// TIA Portal V16 export
// export: Created 2021-11-12T13:32:30.3690276Z, ExportSetting WithDefaults, DisplayName Totally Integrated Automation Portal, DisplayVersion V16 Update 3, DisplayName TIA Portal Version Control Interface, DisplayVersion V16 Update 2, DisplayName TIA Portal Openness, DisplayVersion V16 Update 3, DisplayName SINAMICS Startdrive Advanced, DisplayVersion V16 Update 5, DisplayName SINAMICS Startdrive G130, G150, S120, S150, SINAMICS MV, S210, DisplayVersion V16 Update 5, DisplayName SINAMICS Startdrive G110M, G120, G120C, G120D, G120P, G115D, DisplayVersion V16 Update 5, DisplayName STEP 7 Professional, DisplayVersion V16 Update 3, DisplayName STEP 7 Safety, DisplayVersion V16, DisplayName WinCC UA Professional, DisplayVersion V16 Update 3
FUNCTION_BLOCK "Station 1R4 Seq"   // FB70, LAD
TITLE = Sequence
{ S7_Optimized_Access := 'TRUE' }
VERSION : 0.1
// MICE standard block 
// Sequence
// Block is designed as a template fo creating user sequences
// 
// All temp variables ToChangeXXXX should be replaced or removed.
// 
// Version              Created                        by             Comment
// 0.1                      30. 8. 2018                    PJ           initial version
// stored: AutoNumber true, IsIECCheckEnabled false, IsRetainMemResEnabled false, MemoryReserve 100, SetENOAutomatically false, UDAEnableTagReadback false
   VAR_INPUT
      IS_ZoneM { ExternalAccessible := 'False'; ExternalVisible := 'False'; ExternalWritable := 'False'} : "UDT_Status_main";   // Main structure from zone
      IS_ZoneS { ExternalAccessible := 'False'; ExternalVisible := 'False'; ExternalWritable := 'False'} : "UDT_Zone_Status_specific";   // Specific structure from zone
      IB1EnableSeq : Bool;   // Enable transition of sequence steps.
      IB1Init : Bool;   // Request to initialize sequence
      IB1SetStep : Bool;   // Request to set specific step number
      II_ReqStepNr : UInt;   // Specific step number to be set
      IB1AlmSupp : Bool;   // Alarm suppression - external
      IB1ExtError : Bool;   // External error
   END_VAR
   VAR_OUTPUT
      OS_Status : Struct   // Output status
         Main : "UDT_Status_main";
         Specific : "UDT_Sequence_Status_Specific";
         Error : "UDT_Error01";
      END_STRUCT;
   END_VAR
   VAR_IN_OUT
      XS_Parameter : "UDT_Sequence_Parameter";   // Individual parameter structure
      XS_Command : "UDT_Sequence_Command";   // Individual command structure
   END_VAR
   VAR RETAIN
      SS_Alarm : Struct   // Device alarms
         ExtError : Bool;   // External error / Externí porucha
         StepOvertime : Bool;   // Current step active for too long / Povolená doba trvání kroku překročena
         Res_0_2 : Bool;   // Reserve
         Res_0_3 : Bool;   // Reserve
         Res_0_4 : Bool;   // Reserve
         Res_0_5 : Bool;   // Reserve
         Res_0_6 : Bool;   // Reserve
         Res_0_7 : Bool;   // Reserve
      END_STRUCT;
   END_VAR
   VAR
      SS_Warning : Struct   // Device warnings
         Res : Bool;   // Reserve / Čeká se až bude signál v 1
         Res_1 : Bool;   // Reserve / Čeká se až bude signál v 0
         Res_2 : Bool;   // Reserve / Čeká se až bude signál v 1
         Res_3 : Bool;   // Reserve / Čeká se až bude signál v 0
         Res_4 : Bool;   // Reserve
         Res_5 : Bool;   // Reserve
         Res_6 : Bool;   // Reserve
         Res_7 : Bool;   // Reserve
      END_STRUCT;
      SB1CollErr : Bool;   // Collective error
      SB1CollWrn : Bool;   // Collective warning
   END_VAR
   VAR RETAIN
      SI_ActiveStepNr : UInt;   // Number of active step
   END_VAR
   VAR
      SI_PreviousStepNr : UInt;   // Number of previous step
      ST_TONStepDuration { S7_SetPoint := 'True'} : IEC_TIMER;   // Checking if step is not active for too long.
   END_VAR
   VAR_TEMP
      TS_Parameter : "UDT_Sequence_Parameter";
      TS_Command : "UDT_Sequence_Command";
      TS_Status : Struct
         Main : "UDT_Status_main";
         Specific : "UDT_Sequence_Status_Specific";
         Error : "UDT_Error01";
      END_STRUCT;
      TB1TransitionEnable : Bool;   // Condition from mode enable transition between steps
      TB1AlmSupp : Bool;   // Alarm suppression
      TI_StepTimeIndex : UInt;   // Index to find time for active step.
   END_VAR
   VAR_TEMP   // added for the SCL form of the ladder/FBD networks
      _w1 : Bool;
   END_VAR
BEGIN

REGION Network 1: Clear temporary variables TS_Status - Main, Specific
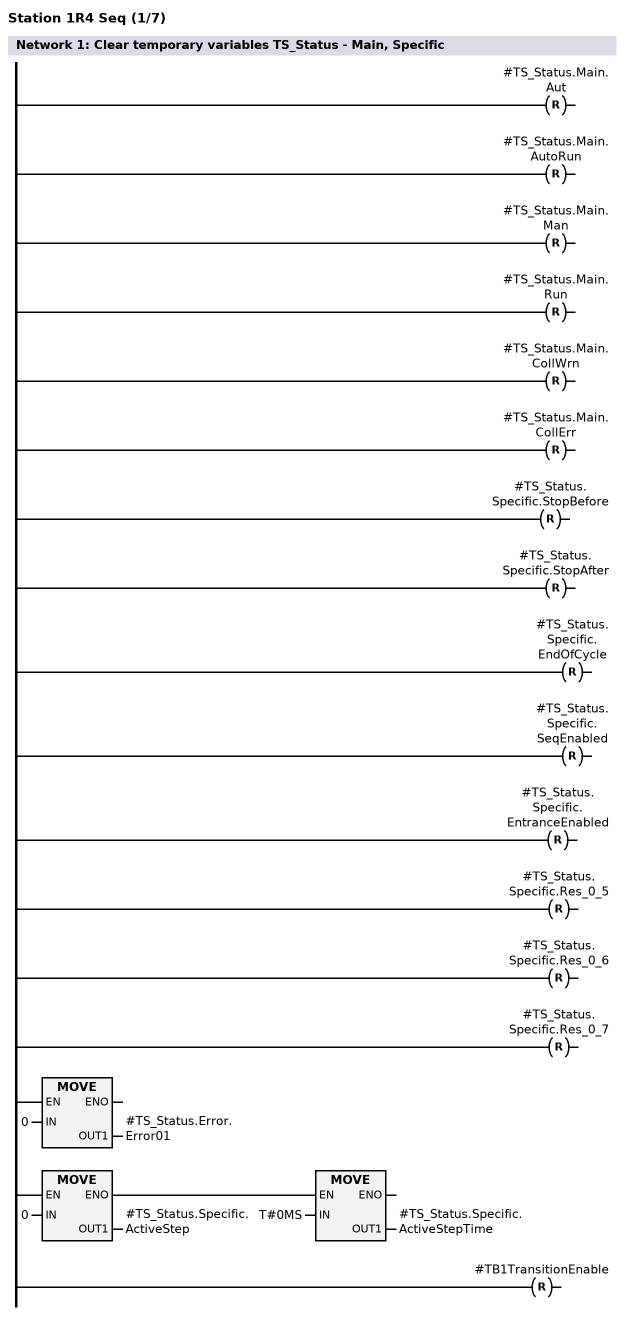
   RUNG wire#powerrail
      R_Coil( #TS_Status.Main.Aut )
   END_RUNG
   RUNG wire#powerrail
      R_Coil( #TS_Status.Main.AutoRun )
   END_RUNG
   RUNG wire#powerrail
      R_Coil( #TS_Status.Main.Man )
   END_RUNG
   RUNG wire#powerrail
      R_Coil( #TS_Status.Main.Run )
   END_RUNG
   RUNG wire#powerrail
      R_Coil( #TS_Status.Main.CollWrn )
   END_RUNG
   RUNG wire#powerrail
      R_Coil( #TS_Status.Main.CollErr )
   END_RUNG
   RUNG wire#powerrail
      R_Coil( #TS_Status.Specific.StopBefore )
   END_RUNG
   RUNG wire#powerrail
      R_Coil( #TS_Status.Specific.StopAfter )
   END_RUNG
   RUNG wire#powerrail
      R_Coil( #TS_Status.Specific.EndOfCycle )
   END_RUNG
   RUNG wire#powerrail
      R_Coil( #TS_Status.Specific.SeqEnabled )
   END_RUNG
   RUNG wire#powerrail
      R_Coil( #TS_Status.Specific.EntranceEnabled )
   END_RUNG
   RUNG wire#powerrail
      R_Coil( #TS_Status.Specific.Res_0_5 )
   END_RUNG
   RUNG wire#powerrail
      R_Coil( #TS_Status.Specific.Res_0_6 )
   END_RUNG
   RUNG wire#powerrail
      R_Coil( #TS_Status.Specific.Res_0_7 )
   END_RUNG
   RUNG wire#powerrail
      Move(in := 0, out1 => #TS_Status.Error.Error01)
   END_RUNG
   RUNG wire#powerrail
      Move(in := 0, out1 => #TS_Status.Specific.ActiveStep)
      Move(in := T#0MS, out1 => #TS_Status.Specific.ActiveStepTime)
   END_RUNG
   RUNG wire#powerrail
      R_Coil( #TB1TransitionEnable )
   END_RUNG
   // the same network as SCL:
   #TS_Status.Main.Aut := FALSE;
   #TS_Status.Main.AutoRun := FALSE;
   #TS_Status.Main.Man := FALSE;
   #TS_Status.Main.Run := FALSE;
   #TS_Status.Main.CollWrn := FALSE;
   #TS_Status.Main.CollErr := FALSE;
   #TS_Status.Specific.StopBefore := FALSE;
   #TS_Status.Specific.StopAfter := FALSE;
   #TS_Status.Specific.EndOfCycle := FALSE;
   #TS_Status.Specific.SeqEnabled := FALSE;
   #TS_Status.Specific.EntranceEnabled := FALSE;
   #TS_Status.Specific.Res_0_5 := FALSE;
   #TS_Status.Specific.Res_0_6 := FALSE;
   #TS_Status.Specific.Res_0_7 := FALSE;
   #TS_Status.Error.Error01 := 0;
   #TS_Status.Specific.ActiveStep := 0;
   #TS_Status.Specific.ActiveStepTime := T#0MS;
   #TB1TransitionEnable := FALSE;
END_REGION

REGION Network 2: Copy In/Out variables to temporary variables
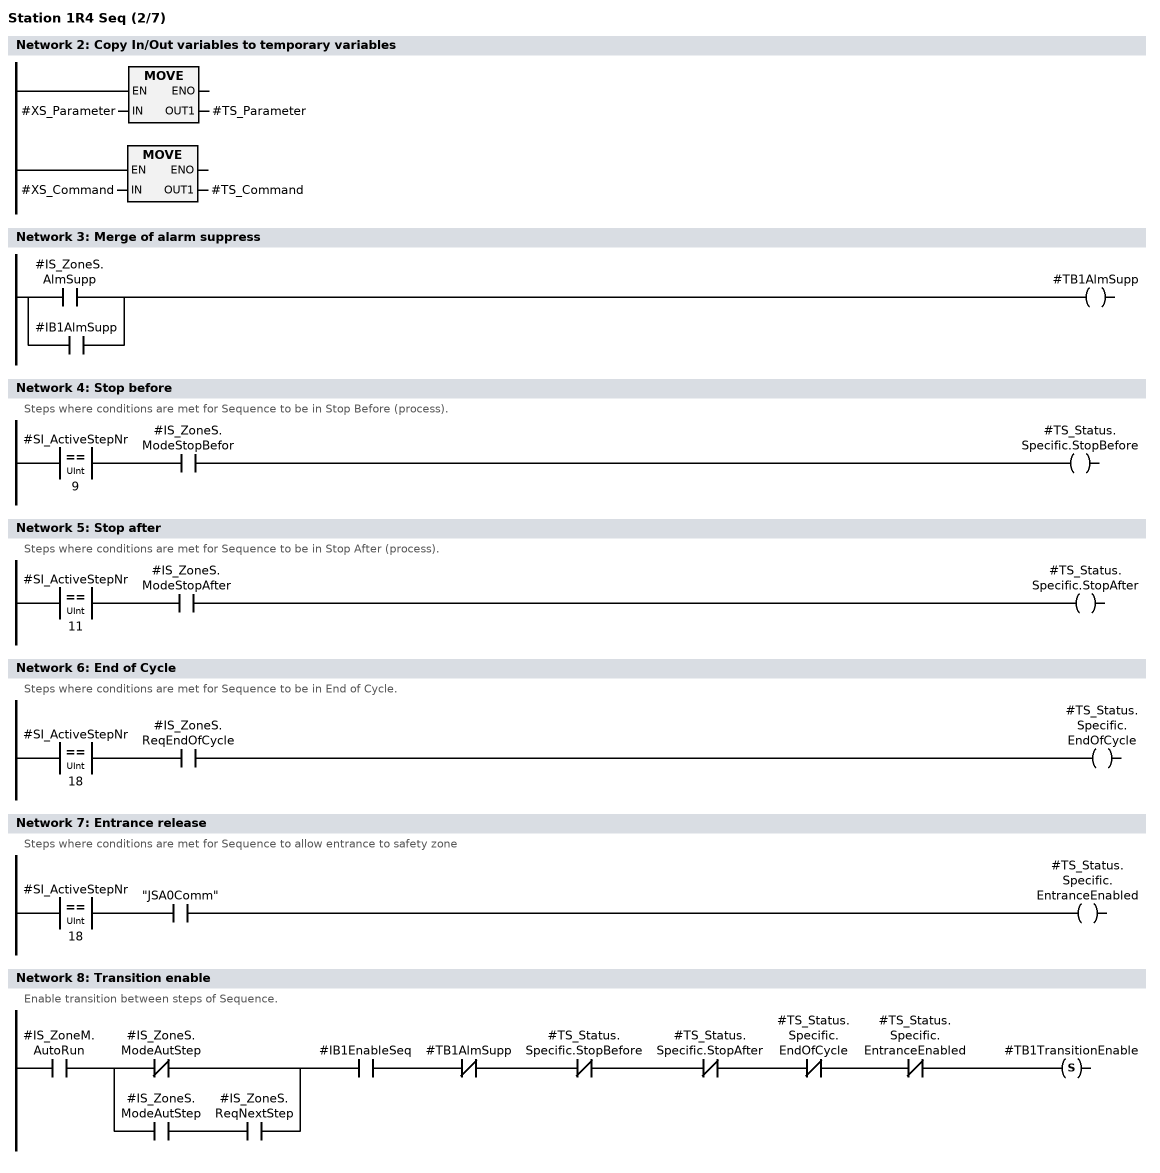
   RUNG wire#powerrail
      Move(in := #XS_Parameter, out1 => #TS_Parameter)
   END_RUNG
   RUNG wire#powerrail
      Move(in := #XS_Command, out1 => #TS_Command)
   END_RUNG
   // the same network as SCL:
   #TS_Parameter := #XS_Parameter;
   #TS_Command := #XS_Command;
END_REGION

REGION Network 3: Merge of alarm suppress
   RUNG wire#powerrail
      Contact( #IS_ZoneS.AlmSupp )
      wire#w1
      Coil( #TB1AlmSupp )
   END_RUNG
   RUNG wire#powerrail
      Contact( #IB1AlmSupp )
   END_RUNG wire#w1
   // the same network as SCL:
   #TB1AlmSupp := #IS_ZoneS.AlmSupp OR #IB1AlmSupp;
END_REGION

REGION Network 4: Stop before
   // Steps where conditions are met for Sequence to be in Stop Before (process).
   RUNG wire#powerrail
      { S7_Templates := "SrcType := UInt" } EQ_Contact(in1 := #SI_ActiveStepNr, in2 := 9)
      Contact( #IS_ZoneS.ModeStopBefor )
      Coil( #TS_Status.Specific.StopBefore )
   END_RUNG
   // the same network as SCL:
   #TS_Status.Specific.StopBefore := (#SI_ActiveStepNr = 9) AND #IS_ZoneS.ModeStopBefor;
END_REGION

REGION Network 5: Stop after
   // Steps where conditions are met for Sequence to be in Stop After (process).
   RUNG wire#powerrail
      { S7_Templates := "SrcType := UInt" } EQ_Contact(in1 := #SI_ActiveStepNr, in2 := 11)
      Contact( #IS_ZoneS.ModeStopAfter )
      Coil( #TS_Status.Specific.StopAfter )
   END_RUNG
   // the same network as SCL:
   #TS_Status.Specific.StopAfter := (#SI_ActiveStepNr = 11) AND #IS_ZoneS.ModeStopAfter;
END_REGION

REGION Network 6: End of Cycle
   // Steps where conditions are met for Sequence to be in End of Cycle.
   RUNG wire#powerrail
      { S7_Templates := "SrcType := UInt" } EQ_Contact(in1 := #SI_ActiveStepNr, in2 := 18)
      Contact( #IS_ZoneS.ReqEndOfCycle )
      Coil( #TS_Status.Specific.EndOfCycle )
   END_RUNG
   // the same network as SCL:
   #TS_Status.Specific.EndOfCycle := (#SI_ActiveStepNr = 18) AND #IS_ZoneS.ReqEndOfCycle;
END_REGION

REGION Network 7: Entrance release
   // Steps where conditions are met for Sequence to allow entrance to safety zone
   RUNG wire#powerrail
      { S7_Templates := "SrcType := UInt" } EQ_Contact(in1 := #SI_ActiveStepNr, in2 := 18)
      Contact( "JSA0Comm" )
      Coil( #TS_Status.Specific.EntranceEnabled )
   END_RUNG
   // the same network as SCL:
   #TS_Status.Specific.EntranceEnabled := (#SI_ActiveStepNr = 18) AND "JSA0Comm";
END_REGION

REGION Network 8: Transition enable
   // Enable transition between steps of Sequence.
   RUNG wire#powerrail
      Contact( #IS_ZoneM.AutoRun )
      wire#w1
      I_Contact( #IS_ZoneS.ModeAutStep )
      wire#w2
      Contact( #IB1EnableSeq )
      I_Contact( #TB1AlmSupp )
      I_Contact( #TS_Status.Specific.StopBefore )
      I_Contact( #TS_Status.Specific.StopAfter )
      I_Contact( #TS_Status.Specific.EndOfCycle )
      I_Contact( #TS_Status.Specific.EntranceEnabled )
      S_Coil( #TB1TransitionEnable )
   END_RUNG
   RUNG wire#w1
      Contact( #IS_ZoneS.ModeAutStep )
      Contact( #IS_ZoneS.ReqNextStep )
   END_RUNG wire#w2
   // the same network as SCL:
   IF #IS_ZoneM.AutoRun AND (NOT #IS_ZoneS.ModeAutStep OR (#IS_ZoneS.ModeAutStep AND #IS_ZoneS.ReqNextStep)) AND #IB1EnableSeq AND NOT #TB1AlmSupp AND NOT #TS_Status.Specific.StopBefore AND NOT #TS_Status.Specific.StopAfter AND NOT #TS_Status.Specific.EndOfCycle AND NOT #TS_Status.Specific.EntranceEnabled THEN
       #TB1TransitionEnable := TRUE;
   END_IF;
END_REGION

REGION Network 9: Init sequence
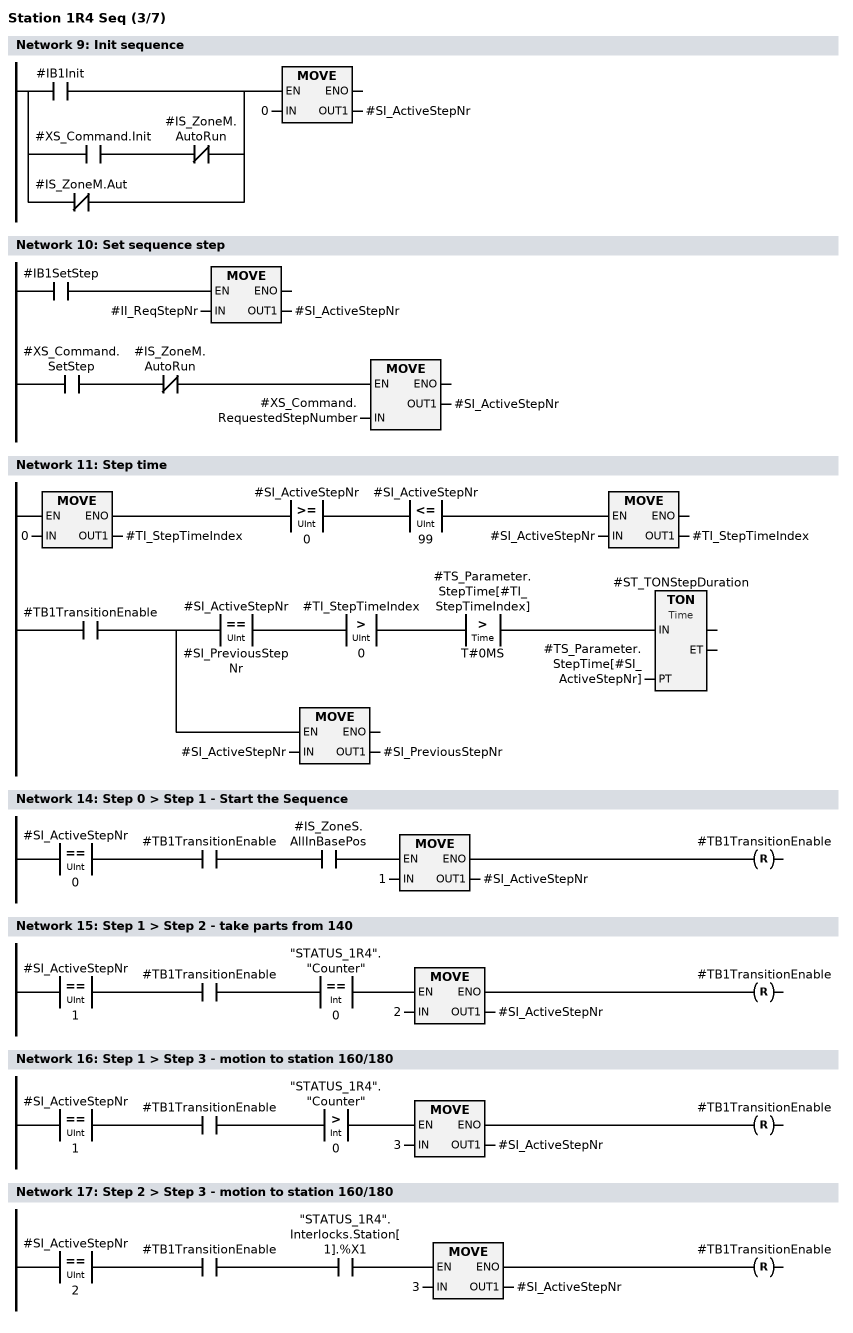
   RUNG wire#powerrail
      Contact( #IB1Init )
      wire#w1
      Move(in := 0, out1 => #SI_ActiveStepNr)
   END_RUNG
   RUNG wire#powerrail
      Contact( #XS_Command.Init )
      I_Contact( #IS_ZoneM.AutoRun )
   END_RUNG wire#w1
   RUNG wire#powerrail
      I_Contact( #IS_ZoneM.Aut )
   END_RUNG wire#w1
   // the same network as SCL:
   IF #IB1Init OR (#XS_Command.Init AND NOT #IS_ZoneM.AutoRun) OR NOT #IS_ZoneM.Aut THEN
       #SI_ActiveStepNr := 0;
   END_IF;
END_REGION

REGION Network 10: Set sequence step
   RUNG wire#powerrail
      Contact( #IB1SetStep )
      Move(in := #II_ReqStepNr, out1 => #SI_ActiveStepNr)
   END_RUNG
   RUNG wire#powerrail
      Contact( #XS_Command.SetStep )
      I_Contact( #IS_ZoneM.AutoRun )
      Move(in := #XS_Command.RequestedStepNumber, out1 => #SI_ActiveStepNr)
   END_RUNG
   // the same network as SCL:
   IF #IB1SetStep THEN #SI_ActiveStepNr := #II_ReqStepNr; END_IF;
   IF #XS_Command.SetStep AND NOT #IS_ZoneM.AutoRun THEN
       #SI_ActiveStepNr := #XS_Command.RequestedStepNumber;
   END_IF;
END_REGION

REGION Network 11: Step time
   RUNG wire#powerrail
      Move(in := 0, out1 => #TI_StepTimeIndex)
      { S7_Templates := "SrcType := UInt" } GE_Contact(in1 := #SI_ActiveStepNr, in2 := 0)
      { S7_Templates := "SrcType := UInt" } LE_Contact(in1 := #SI_ActiveStepNr, in2 := 99)
      Move(in := #SI_ActiveStepNr, out1 => #TI_StepTimeIndex)
   END_RUNG
   RUNG wire#powerrail
      Contact( #TB1TransitionEnable )
      wire#w1
      { S7_Templates := "SrcType := UInt" } EQ_Contact(in1 := #SI_ActiveStepNr, in2 := #SI_PreviousStepNr)
      { S7_Templates := "SrcType := UInt" } GT_Contact(in1 := #TI_StepTimeIndex, in2 := 0)
      { S7_Templates := "SrcType := Time" } GT_Contact(in1 := #TS_Parameter.StepTime[#TI_StepTimeIndex], in2 := T#0MS)
      { S7_Templates := "time_type := Time" } #ST_TONStepDuration.TON(pt := #TS_Parameter.StepTime[#SI_ActiveStepNr], et =>)
   END_RUNG
   RUNG wire#w1
      Move(in := #SI_ActiveStepNr, out1 => #SI_PreviousStepNr)
   END_RUNG
   // the same network as SCL:
   #TI_StepTimeIndex := 0;
   IF (#SI_ActiveStepNr >= 0) AND (#SI_ActiveStepNr <= 99) THEN
       #TI_StepTimeIndex := #SI_ActiveStepNr;
   END_IF;
   #ST_TONStepDuration.TON(IN := #TB1TransitionEnable AND (#SI_ActiveStepNr = #SI_PreviousStepNr) AND (#TI_StepTimeIndex > 0) AND (#TS_Parameter.StepTime[#TI_StepTimeIndex] > T#0MS),
                           PT := #TS_Parameter.StepTime[#SI_ActiveStepNr]);
   IF #TB1TransitionEnable THEN #SI_PreviousStepNr := #SI_ActiveStepNr; END_IF;
END_REGION

REGION Network 12: Operator info status
END_REGION

REGION Network 13: *************** Sequence steps ***********************
   // No parallel conditions. If neccessary > for each condition its own network (Active step / conditions / step change). This also solves jumps.
   // No "active" parts in step. So no timers, counters, comparators etc. those belong to Creating conditions section or outside this block. Only simple bool conditions.
   // Always reset TB1_TransitionEnable bit. This will make sure on PLC cycle only one step of sequence will be processed.
   // Last step/network should be that if active step number is bigger then last used one go to zero step.
END_REGION

REGION Network 14: Step 0 > Step 1 - Start the Sequence
   RUNG wire#powerrail
      { S7_Templates := "SrcType := UInt" } EQ_Contact(in1 := #SI_ActiveStepNr, in2 := 0)
      Contact( #TB1TransitionEnable )
      Contact( #IS_ZoneS.AllInBasePos )
      Move(in := 1, out1 => #SI_ActiveStepNr)
      R_Coil( #TB1TransitionEnable )
   END_RUNG
   // the same network as SCL:
   #_w1 := (#SI_ActiveStepNr = 0) AND #TB1TransitionEnable AND #IS_ZoneS.AllInBasePos;
   IF #_w1 THEN
       #SI_ActiveStepNr := 1;
       #TB1TransitionEnable := FALSE;
   END_IF;
END_REGION

REGION Network 15: Step 1 > Step 2 - take parts from 140
   RUNG wire#powerrail
      { S7_Templates := "SrcType := UInt" } EQ_Contact(in1 := #SI_ActiveStepNr, in2 := 1)
      Contact( #TB1TransitionEnable )
      { S7_Templates := "SrcType := Int" } EQ_Contact(in1 := "STATUS_1R4"."Counter", in2 := 0)
      Move(in := 2, out1 => #SI_ActiveStepNr)
      R_Coil( #TB1TransitionEnable )
   END_RUNG
   // the same network as SCL:
   #_w1 := (#SI_ActiveStepNr = 1) AND #TB1TransitionEnable AND ("STATUS_1R4"."Counter" = 0);
   IF #_w1 THEN
       #SI_ActiveStepNr := 2;
       #TB1TransitionEnable := FALSE;
   END_IF;
END_REGION

REGION Network 16: Step 1 > Step 3 - motion to station 160/180
   RUNG wire#powerrail
      { S7_Templates := "SrcType := UInt" } EQ_Contact(in1 := #SI_ActiveStepNr, in2 := 1)
      Contact( #TB1TransitionEnable )
      { S7_Templates := "SrcType := Int" } GT_Contact(in1 := "STATUS_1R4"."Counter", in2 := 0)
      Move(in := 3, out1 => #SI_ActiveStepNr)
      R_Coil( #TB1TransitionEnable )
   END_RUNG
   // the same network as SCL:
   #_w1 := (#SI_ActiveStepNr = 1) AND #TB1TransitionEnable AND ("STATUS_1R4"."Counter" > 0);
   IF #_w1 THEN
       #SI_ActiveStepNr := 3;
       #TB1TransitionEnable := FALSE;
   END_IF;
END_REGION

REGION Network 17: Step 2 > Step 3 - motion to station 160/180
   RUNG wire#powerrail
      { S7_Templates := "SrcType := UInt" } EQ_Contact(in1 := #SI_ActiveStepNr, in2 := 2)
      Contact( #TB1TransitionEnable )
      Contact( "STATUS_1R4".Interlocks.Station[1].%X1 )
      Move(in := 3, out1 => #SI_ActiveStepNr)
      R_Coil( #TB1TransitionEnable )
   END_RUNG
   // the same network as SCL:
   #_w1 := (#SI_ActiveStepNr = 2) AND #TB1TransitionEnable AND "STATUS_1R4".Interlocks.Station[1].%X1;
   IF #_w1 THEN
       #SI_ActiveStepNr := 3;
       #TB1TransitionEnable := FALSE;
   END_IF;
END_REGION

REGION Network 18: Step 3 > Step 4 - put parts to station 160 / 180
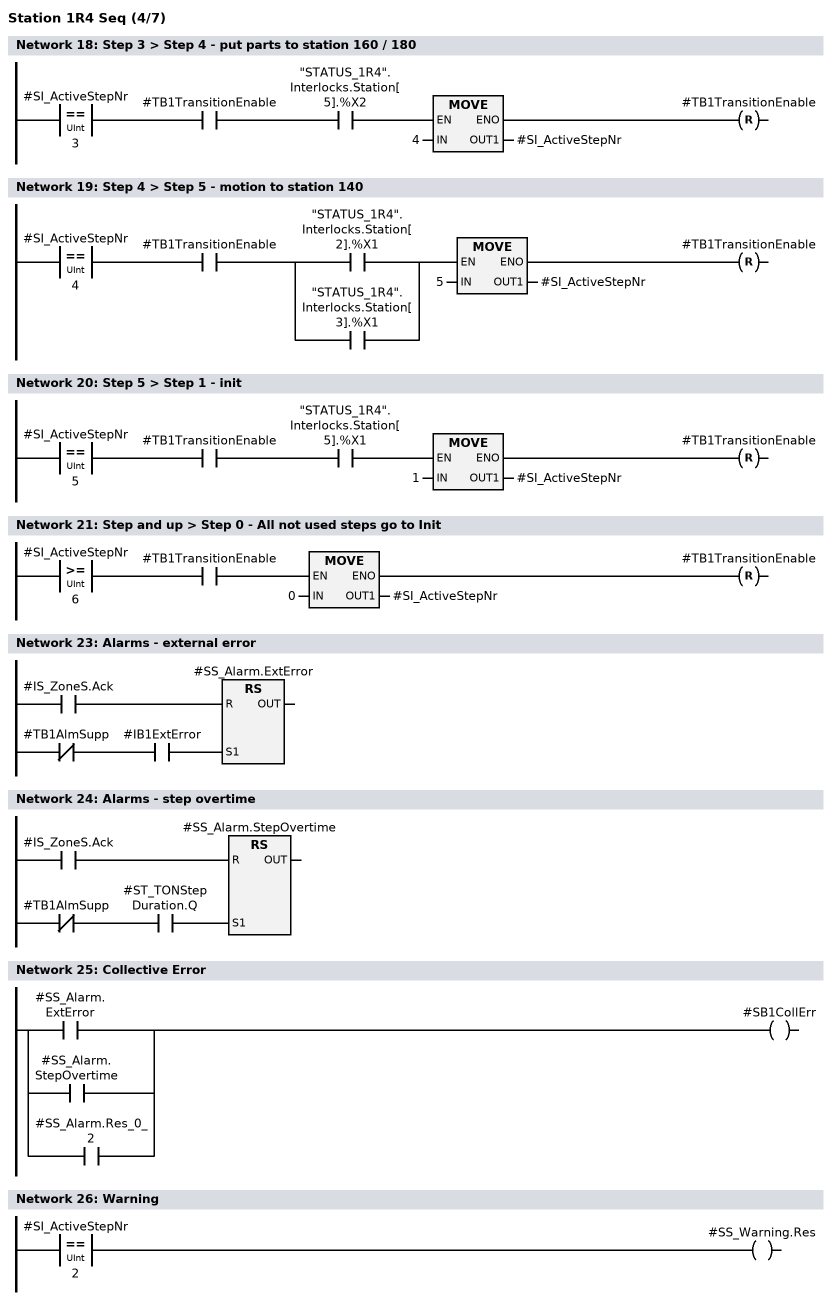
   RUNG wire#powerrail
      { S7_Templates := "SrcType := UInt" } EQ_Contact(in1 := #SI_ActiveStepNr, in2 := 3)
      Contact( #TB1TransitionEnable )
      Contact( "STATUS_1R4".Interlocks.Station[5].%X2 )
      Move(in := 4, out1 => #SI_ActiveStepNr)
      R_Coil( #TB1TransitionEnable )
   END_RUNG
   // the same network as SCL:
   #_w1 := (#SI_ActiveStepNr = 3) AND #TB1TransitionEnable AND "STATUS_1R4".Interlocks.Station[5].%X2;
   IF #_w1 THEN
       #SI_ActiveStepNr := 4;
       #TB1TransitionEnable := FALSE;
   END_IF;
END_REGION

REGION Network 19: Step 4 > Step 5 - motion to station 140
   RUNG wire#powerrail
      { S7_Templates := "SrcType := UInt" } EQ_Contact(in1 := #SI_ActiveStepNr, in2 := 4)
      Contact( #TB1TransitionEnable )
      wire#w1
      Contact( "STATUS_1R4".Interlocks.Station[2].%X1 )
      wire#w2
      Move(in := 5, out1 => #SI_ActiveStepNr)
      R_Coil( #TB1TransitionEnable )
   END_RUNG
   RUNG wire#w1
      Contact( "STATUS_1R4".Interlocks.Station[3].%X1 )
   END_RUNG wire#w2
   // the same network as SCL:
   #_w1 := (#SI_ActiveStepNr = 4) AND #TB1TransitionEnable AND ("STATUS_1R4".Interlocks.Station[2].%X1 OR "STATUS_1R4".Interlocks.Station[3].%X1);
   IF #_w1 THEN
       #SI_ActiveStepNr := 5;
       #TB1TransitionEnable := FALSE;
   END_IF;
END_REGION

REGION Network 20: Step 5 > Step 1 - init
   RUNG wire#powerrail
      { S7_Templates := "SrcType := UInt" } EQ_Contact(in1 := #SI_ActiveStepNr, in2 := 5)
      Contact( #TB1TransitionEnable )
      Contact( "STATUS_1R4".Interlocks.Station[5].%X1 )
      Move(in := 1, out1 => #SI_ActiveStepNr)
      R_Coil( #TB1TransitionEnable )
   END_RUNG
   // the same network as SCL:
   #_w1 := (#SI_ActiveStepNr = 5) AND #TB1TransitionEnable AND "STATUS_1R4".Interlocks.Station[5].%X1;
   IF #_w1 THEN
       #SI_ActiveStepNr := 1;
       #TB1TransitionEnable := FALSE;
   END_IF;
END_REGION

REGION Network 21: Step and up > Step 0 - All not used steps go to Init
   RUNG wire#powerrail
      { S7_Templates := "SrcType := UInt" } GE_Contact(in1 := #SI_ActiveStepNr, in2 := 6)
      Contact( #TB1TransitionEnable )
      Move(in := 0, out1 => #SI_ActiveStepNr)
      R_Coil( #TB1TransitionEnable )
   END_RUNG
   // the same network as SCL:
   #_w1 := (#SI_ActiveStepNr >= 6) AND #TB1TransitionEnable;
   IF #_w1 THEN
       #SI_ActiveStepNr := 0;
       #TB1TransitionEnable := FALSE;
   END_IF;
END_REGION

REGION Network 22: *************** Alarm and warning section ***********************
END_REGION

REGION Network 23: Alarms - external error
   RUNG wire#powerrail
      Contact( #IS_ZoneS.Ack )
      S_RS(operand := #SS_Alarm.ExtError, s1 := wire#w1)
   END_RUNG
   RUNG wire#powerrail
      I_Contact( #TB1AlmSupp )
      Contact( #IB1ExtError )
   END_RUNG wire#w1
   // the same network as SCL:
   IF #IS_ZoneS.Ack THEN
       #SS_Alarm.ExtError := FALSE;   // RS flip-flop
   END_IF;
   IF NOT #TB1AlmSupp AND #IB1ExtError THEN #SS_Alarm.ExtError := TRUE; END_IF;
END_REGION

REGION Network 24: Alarms - step overtime
   RUNG wire#powerrail
      Contact( #IS_ZoneS.Ack )
      S_RS(operand := #SS_Alarm.StepOvertime, s1 := wire#w1)
   END_RUNG
   RUNG wire#powerrail
      I_Contact( #TB1AlmSupp )
      Contact( #ST_TONStepDuration.Q )
   END_RUNG wire#w1
   // the same network as SCL:
   IF #IS_ZoneS.Ack THEN
       #SS_Alarm.StepOvertime := FALSE;   // RS flip-flop
   END_IF;
   IF NOT #TB1AlmSupp AND #ST_TONStepDuration.Q THEN #SS_Alarm.StepOvertime := TRUE; END_IF;
END_REGION

REGION Network 25: Collective Error
   RUNG wire#powerrail
      Contact( #SS_Alarm.ExtError )
      wire#w1
      Coil( #SB1CollErr )
   END_RUNG
   RUNG wire#powerrail
      Contact( #SS_Alarm.StepOvertime )
   END_RUNG wire#w1
   RUNG wire#powerrail
      Contact( #SS_Alarm.Res_0_2 )
   END_RUNG wire#w1
   // the same network as SCL:
   #SB1CollErr := #SS_Alarm.ExtError OR #SS_Alarm.StepOvertime OR #SS_Alarm.Res_0_2;
END_REGION

REGION Network 26: Warning
   RUNG wire#powerrail
      { S7_Templates := "SrcType := UInt" } EQ_Contact(in1 := #SI_ActiveStepNr, in2 := 2)
      Coil( #SS_Warning.Res )
   END_RUNG
   // the same network as SCL:
   #SS_Warning.Res := #SI_ActiveStepNr = 2;
END_REGION

REGION Network 27: Collective Warning
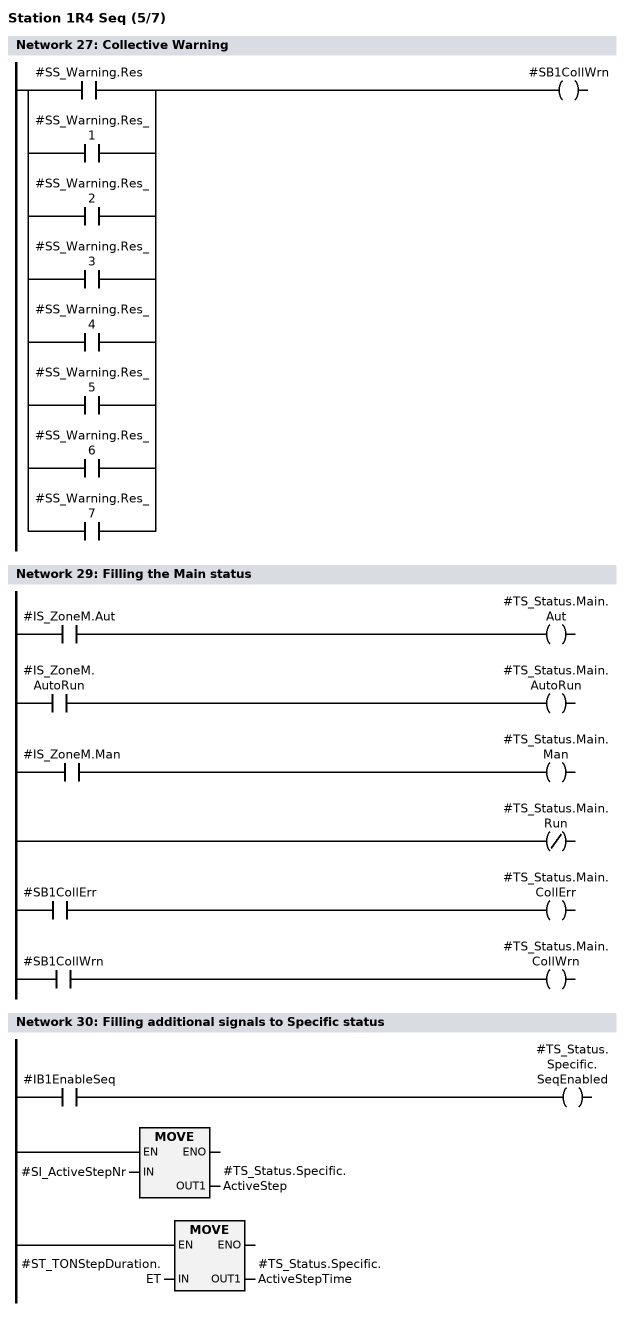
   RUNG wire#powerrail
      Contact( #SS_Warning.Res )
      wire#w1
      Coil( #SB1CollWrn )
   END_RUNG
   RUNG wire#powerrail
      Contact( #SS_Warning.Res_1 )
   END_RUNG wire#w1
   RUNG wire#powerrail
      Contact( #SS_Warning.Res_2 )
   END_RUNG wire#w1
   RUNG wire#powerrail
      Contact( #SS_Warning.Res_3 )
   END_RUNG wire#w1
   RUNG wire#powerrail
      Contact( #SS_Warning.Res_4 )
   END_RUNG wire#w1
   RUNG wire#powerrail
      Contact( #SS_Warning.Res_5 )
   END_RUNG wire#w1
   RUNG wire#powerrail
      Contact( #SS_Warning.Res_6 )
   END_RUNG wire#w1
   RUNG wire#powerrail
      Contact( #SS_Warning.Res_7 )
   END_RUNG wire#w1
   // the same network as SCL:
   #SB1CollWrn := #SS_Warning.Res OR #SS_Warning.Res_1 OR #SS_Warning.Res_2 OR #SS_Warning.Res_3 OR #SS_Warning.Res_4 OR #SS_Warning.Res_5 OR #SS_Warning.Res_6 OR #SS_Warning.Res_7;
END_REGION

REGION Network 28: *************** Fill out structures / Copy to outputs ***********************
END_REGION

REGION Network 29: Filling the Main status
   RUNG wire#powerrail
      Contact( #IS_ZoneM.Aut )
      Coil( #TS_Status.Main.Aut )
   END_RUNG
   RUNG wire#powerrail
      Contact( #IS_ZoneM.AutoRun )
      Coil( #TS_Status.Main.AutoRun )
   END_RUNG
   RUNG wire#powerrail
      Contact( #IS_ZoneM.Man )
      Coil( #TS_Status.Main.Man )
   END_RUNG
   RUNG wire#powerrail
      I_Coil( #TS_Status.Main.Run )
   END_RUNG
   RUNG wire#powerrail
      Contact( #SB1CollErr )
      Coil( #TS_Status.Main.CollErr )
   END_RUNG
   RUNG wire#powerrail
      Contact( #SB1CollWrn )
      Coil( #TS_Status.Main.CollWrn )
   END_RUNG
   // the same network as SCL:
   #TS_Status.Main.Aut := #IS_ZoneM.Aut;
   #TS_Status.Main.AutoRun := #IS_ZoneM.AutoRun;
   #TS_Status.Main.Man := #IS_ZoneM.Man;
   #TS_Status.Main.Run := NOT TRUE;
   #TS_Status.Main.CollErr := #SB1CollErr;
   #TS_Status.Main.CollWrn := #SB1CollWrn;
END_REGION

REGION Network 30: Filling additional signals to Specific status
   RUNG wire#powerrail
      Contact( #IB1EnableSeq )
      Coil( #TS_Status.Specific.SeqEnabled )
   END_RUNG
   RUNG wire#powerrail
      Move(in := #SI_ActiveStepNr, out1 => #TS_Status.Specific.ActiveStep)
   END_RUNG
   RUNG wire#powerrail
      Move(in := #ST_TONStepDuration.ET, out1 => #TS_Status.Specific.ActiveStepTime)
   END_RUNG
   // the same network as SCL:
   #TS_Status.Specific.SeqEnabled := #IB1EnableSeq;
   #TS_Status.Specific.ActiveStep := #SI_ActiveStepNr;
   #TS_Status.Specific.ActiveStepTime := #ST_TONStepDuration.ET;
END_REGION

REGION Network 31: Reset commands
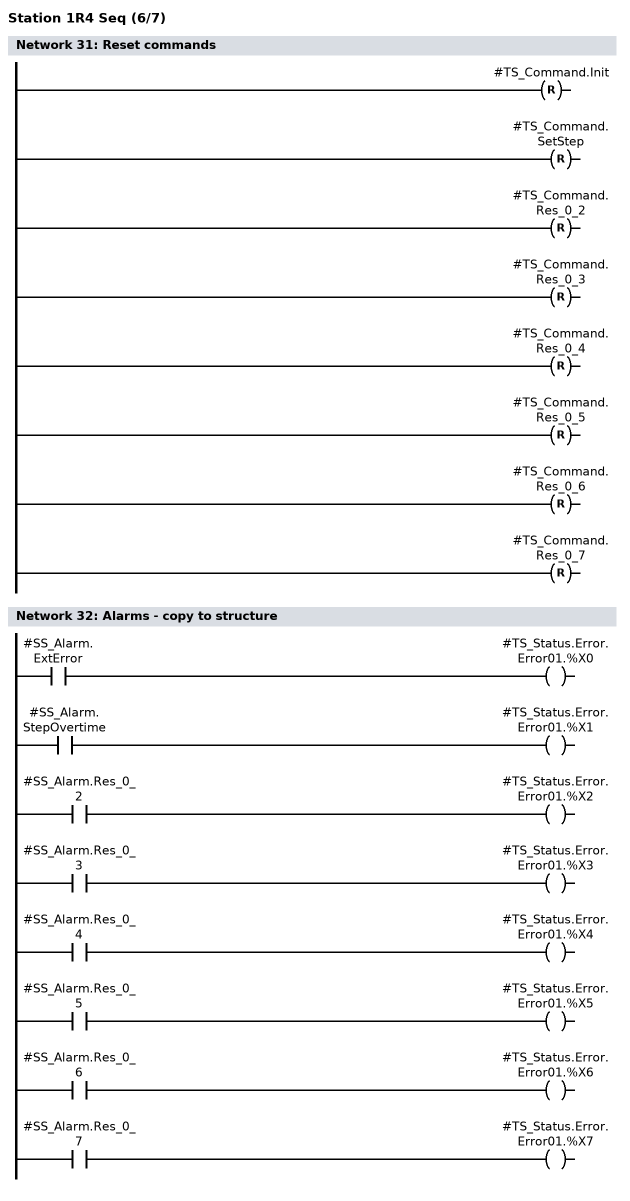
   RUNG wire#powerrail
      R_Coil( #TS_Command.Init )
   END_RUNG
   RUNG wire#powerrail
      R_Coil( #TS_Command.SetStep )
   END_RUNG
   RUNG wire#powerrail
      R_Coil( #TS_Command.Res_0_2 )
   END_RUNG
   RUNG wire#powerrail
      R_Coil( #TS_Command.Res_0_3 )
   END_RUNG
   RUNG wire#powerrail
      R_Coil( #TS_Command.Res_0_4 )
   END_RUNG
   RUNG wire#powerrail
      R_Coil( #TS_Command.Res_0_5 )
   END_RUNG
   RUNG wire#powerrail
      R_Coil( #TS_Command.Res_0_6 )
   END_RUNG
   RUNG wire#powerrail
      R_Coil( #TS_Command.Res_0_7 )
   END_RUNG
   // the same network as SCL:
   #TS_Command.Init := FALSE;
   #TS_Command.SetStep := FALSE;
   #TS_Command.Res_0_2 := FALSE;
   #TS_Command.Res_0_3 := FALSE;
   #TS_Command.Res_0_4 := FALSE;
   #TS_Command.Res_0_5 := FALSE;
   #TS_Command.Res_0_6 := FALSE;
   #TS_Command.Res_0_7 := FALSE;
END_REGION

REGION Network 32: Alarms - copy to structure
   RUNG wire#powerrail
      Contact( #SS_Alarm.ExtError )
      Coil( #TS_Status.Error.Error01.%X0 )
   END_RUNG
   RUNG wire#powerrail
      Contact( #SS_Alarm.StepOvertime )
      Coil( #TS_Status.Error.Error01.%X1 )
   END_RUNG
   RUNG wire#powerrail
      Contact( #SS_Alarm.Res_0_2 )
      Coil( #TS_Status.Error.Error01.%X2 )
   END_RUNG
   RUNG wire#powerrail
      Contact( #SS_Alarm.Res_0_3 )
      Coil( #TS_Status.Error.Error01.%X3 )
   END_RUNG
   RUNG wire#powerrail
      Contact( #SS_Alarm.Res_0_4 )
      Coil( #TS_Status.Error.Error01.%X4 )
   END_RUNG
   RUNG wire#powerrail
      Contact( #SS_Alarm.Res_0_5 )
      Coil( #TS_Status.Error.Error01.%X5 )
   END_RUNG
   RUNG wire#powerrail
      Contact( #SS_Alarm.Res_0_6 )
      Coil( #TS_Status.Error.Error01.%X6 )
   END_RUNG
   RUNG wire#powerrail
      Contact( #SS_Alarm.Res_0_7 )
      Coil( #TS_Status.Error.Error01.%X7 )
   END_RUNG
   // the same network as SCL:
   #TS_Status.Error.Error01.%X0 := #SS_Alarm.ExtError;
   #TS_Status.Error.Error01.%X1 := #SS_Alarm.StepOvertime;
   #TS_Status.Error.Error01.%X2 := #SS_Alarm.Res_0_2;
   #TS_Status.Error.Error01.%X3 := #SS_Alarm.Res_0_3;
   #TS_Status.Error.Error01.%X4 := #SS_Alarm.Res_0_4;
   #TS_Status.Error.Error01.%X5 := #SS_Alarm.Res_0_5;
   #TS_Status.Error.Error01.%X6 := #SS_Alarm.Res_0_6;
   #TS_Status.Error.Error01.%X7 := #SS_Alarm.Res_0_7;
END_REGION

REGION Network 33: Warnings - copy to structure
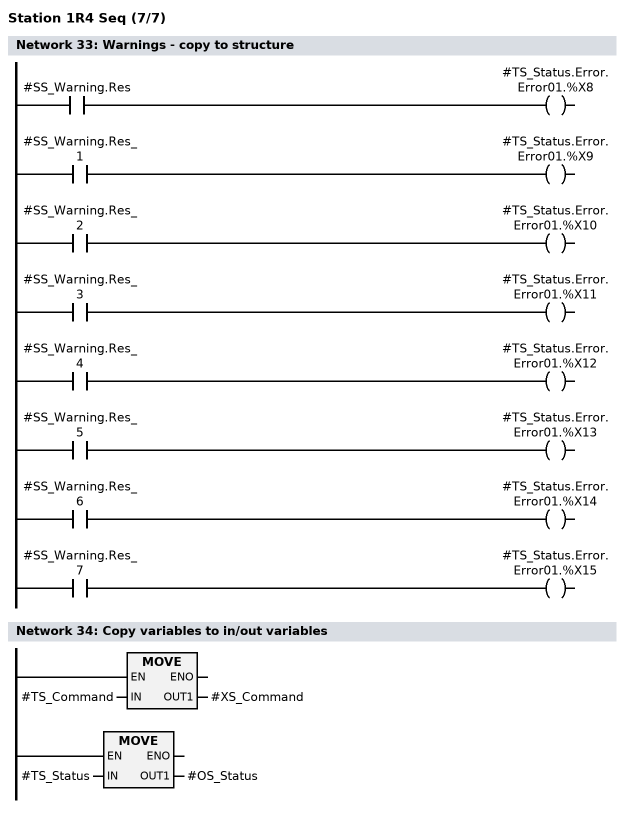
   RUNG wire#powerrail
      Contact( #SS_Warning.Res )
      Coil( #TS_Status.Error.Error01.%X8 )
   END_RUNG
   RUNG wire#powerrail
      Contact( #SS_Warning.Res_1 )
      Coil( #TS_Status.Error.Error01.%X9 )
   END_RUNG
   RUNG wire#powerrail
      Contact( #SS_Warning.Res_2 )
      Coil( #TS_Status.Error.Error01.%X10 )
   END_RUNG
   RUNG wire#powerrail
      Contact( #SS_Warning.Res_3 )
      Coil( #TS_Status.Error.Error01.%X11 )
   END_RUNG
   RUNG wire#powerrail
      Contact( #SS_Warning.Res_4 )
      Coil( #TS_Status.Error.Error01.%X12 )
   END_RUNG
   RUNG wire#powerrail
      Contact( #SS_Warning.Res_5 )
      Coil( #TS_Status.Error.Error01.%X13 )
   END_RUNG
   RUNG wire#powerrail
      Contact( #SS_Warning.Res_6 )
      Coil( #TS_Status.Error.Error01.%X14 )
   END_RUNG
   RUNG wire#powerrail
      Contact( #SS_Warning.Res_7 )
      Coil( #TS_Status.Error.Error01.%X15 )
   END_RUNG
   // the same network as SCL:
   #TS_Status.Error.Error01.%X8 := #SS_Warning.Res;
   #TS_Status.Error.Error01.%X9 := #SS_Warning.Res_1;
   #TS_Status.Error.Error01.%X10 := #SS_Warning.Res_2;
   #TS_Status.Error.Error01.%X11 := #SS_Warning.Res_3;
   #TS_Status.Error.Error01.%X12 := #SS_Warning.Res_4;
   #TS_Status.Error.Error01.%X13 := #SS_Warning.Res_5;
   #TS_Status.Error.Error01.%X14 := #SS_Warning.Res_6;
   #TS_Status.Error.Error01.%X15 := #SS_Warning.Res_7;
END_REGION

REGION Network 34: Copy variables to in/out variables
   RUNG wire#powerrail
      Move(in := #TS_Command, out1 => #XS_Command)
   END_RUNG
   RUNG wire#powerrail
      Move(in := #TS_Status, out1 => #OS_Status)
   END_RUNG
   // the same network as SCL:
   #XS_Command := #TS_Command;
   #OS_Status := #TS_Status;
END_REGION
END_FUNCTION_BLOCK
